// TIA Portal V16 export
// export: Created 2021-07-12T14:47:20.3088612Z, ExportSetting WithDefaults, DisplayName Totally Integrated Automation Portal, DisplayVersion V16, DisplayName TIA Portal Version Control Interface, DisplayVersion V16, DisplayName TIA Portal Openness, DisplayVersion V16, DisplayName STEP 7 Professional, DisplayVersion V16, DisplayName STEP 7 Safety, DisplayVersion V16, DisplayName WinCC Professional, DisplayVersion V16
TYPE "SimaHydTO_typeHMIConnectionAxisSelectorStatus"
TITLE = SimaHydTO_typeHMIConnectionAxisSelectorStatus
// HMI interface: Axis selection of axis array - Status (PLC -> HMI)
// stored: IsFailsafeCompliant false
   STRUCT
      actualAxisIndex : Int;   // Actual selected array index
      selectedAxis : DB_ANY;   // DB number of actual selected hydraulic axis
      selectedTO_Axis : DB_ANY;   // DB/TO number of actual selected technology object axis
      selectedVChar : DB_ANY;   // DB number of actual selected valve characteristics
      selectedAxisInteger : UInt;   // DB number of actual selected hydraulic axis as integer value
      selectedAxisTOInteger : UInt;   // DB/TO number of actual selected technology object as integer value
      selectedVCharInteger : UInt;   // DB number of actual selected valve characteristics as integer value
      selectedAxisName : WString[24];   // Name of actual selected hydraulic axis
      selectedVCharName : WString[24];   // Name of active VChat of selected hydraulic axis
      selectedTypeOfAxis : Int;   // 0: No axis / 1: Speed axis / 2: Positioning axis / 3: Synchronous axis / 4: External encoder
      selectionChanged : Bool;   // axis selection is changed
      dataValid : Bool;   // Selected data valid
      dataError : Bool;   // Error of data selection
   END_STRUCT;
END_TYPE
